FUNCTION_BLOCK AX_D_FF (* Data latch (d) flip flop *)
  (* Standard: 61499-1 Annex A; Description: Copyright (c) 2017 fortiss GmbH This program and the accompanying materials are made available under the terms of the Eclipse Public License 2.0 which is available at https://www.eclipse.org/legal/epl-2.0/ SPDX-License-Identifier: EPL-2.0 *)
  (* Version 3.0, 2025-04-14, Patrick Aigner, changed package *)
  (* Version 1.0, 2017-09-22, Alois Zoitl, fortiss GmbH, initial API and implementation and/or initial documentation *)
  PACKAGE adapter::events::unidirectional;
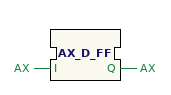
  SOCKETS
    I : adapter::types::unidirectional::AX; (* Value to latch *)
  END_SOCKETS
  PLUGS
    Q : adapter::types::unidirectional::AX; (* Latched value *)
  END_PLUGS
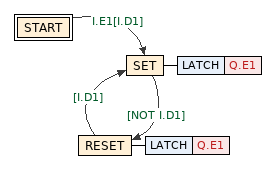
  EC_STATES
    START; (* Initial State *)
    SET : LATCH -> Q.E1; (* Initialization *)
    RESET : LATCH -> Q.E1;
  END_STATES
  EC_TRANSITIONS
    START TO SET := I.E1[I.D1];
    SET TO RESET := [NOT I.D1];
    RESET TO SET := [I.D1];
  END_TRANSITIONS
  ALGORITHM LATCH IN ST:
Q.D1 := I.D1;
  END_ALGORITHM
END_FUNCTION_BLOCK
